Yaskawa INFORM job: KRIS_OTHER_WELDS.JBI

/JOB
//NAME KRIS_OTHER_WELDS
//POS
///NPOS 371,371,371,14,0,0
///TOOL 0
///POSTYPE PULSE
///PULSE
C00000=36471,-76527,-106813,-19264,71481,-77238
C00001=66631,50103,-4762,13566,84527,65375
C00002=104392,-45604,-45068,41730,67848,43971
C00003=102772,-23592,-15673,48581,65359,41958
C00004=103105,-4521,-1193,48225,65783,42370
C00005=103550,-365,5452,48799,64222,41754
C00006=103550,625,8518,49296,63299,41230
C00007=103550,355,7706,49163,63541,41368
C00008=102300,1028,8270,49380,64218,41057
C00009=102134,1217,8640,49454,64220,40967
C00010=102487,1102,8722,49434,63955,41010
C00011=101792,827,6993,49227,64947,41190
C00012=100819,-958,-818,48185,68095,42388
C00013=74228,-100728,-57385,53918,72446,30220
C00014=60504,-146661,-111893,16693,92041,-63510
C00015=81002,-144165,-111893,31958,74905,-63510
C00016=99609,-128801,-101652,29194,69226,-57515
C00017=99609,-127984,-100239,29275,68831,-57620
C00018=99609,-128289,-100766,29244,68978,-57581
C00019=102150,-129321,-101059,28822,67791,-56859
C00020=99944,-132310,-102446,29373,67957,-57721
C00021=94854,-157221,-110079,32013,62771,-61374
C00022=94854,-157221,-110079,32013,62771,-61374
C00023=150575,-180894,-113467,-20602,37776,7473
C00024=131435,-154210,-106652,-7413,43941,-3112
C00025=131414,-154056,-106648,-7392,44016,-3129
C00026=131048,-150684,-105922,-7028,45259,-3400
C00027=131414,-154056,-106648,-7392,44016,-3129
C00028=178670,-106537,-94441,-32173,86364,27351
C00029=174579,-86120,-85943,-32864,94727,28981
C00030=173469,-85635,-85233,-32803,94141,28710
C00031=173469,-85539,-84108,-32766,93596,28870
C00032=173084,-86046,-85408,-32780,93905,28625
C00033=171779,-87936,-86208,-32689,92999,28371
C00034=172551,-86827,-85740,-32743,93534,28522
C00035=185237,-110424,-94728,-32531,92831,33795
C00036=185237,-110424,-94728,-32531,92831,33795
C00037=134012,-175619,-118342,2096,46955,-2797
C00038=133371,-126486,-107062,2327,67886,-2658
C00039=134292,-123400,-104700,2048,67993,-2322
C00040=134292,-122480,-102592,2060,67168,-2335
C00041=134292,-122828,-103379,2055,67474,-2331
C00042=133740,-117277,-101631,2195,69264,-2498
C00043=134292,-122828,-103379,2055,67474,-2331
C00044=145565,-124760,-104669,-1363,67226,1769
C00045=157884,-133264,-102216,-16015,55602,12124
C00046=154931,-135462,-102806,-14939,54301,11078
C00047=159722,-139649,-104449,-17130,54142,13140
C00048=121501,-151260,-116369,16790,67529,-22254
C00049=84851,-125920,-106326,14509,72614,-18670
C00050=87302,-113526,-101119,13757,75261,-17475
C00051=88050,-112106,-100360,13572,75391,-17193
C00052=88050,-111725,-99039,13608,74790,-17261
C00053=88050,-111984,-99928,13584,75193,-17215
C00054=88832,-108808,-98834,13352,75998,-16846
C00055=87807,-112947,-100252,13656,74947,-17329
C00056=92070,-142291,-103311,16392,49176,-14760
C00057=94804,-140634,-102905,14943,49236,-13516
C00058=91121,-138706,-102421,16531,50612,-14939
C00059=93561,-140381,-102567,15560,49394,-14049
C00060=69173,-195704,-118009,34153,38892,-29324
C00061=69173,-195704,-118009,34153,38892,-29324
C00062=107696,-37154,-67359,5229,84713,-5863
C00063=116742,-32674,-55171,12076,80004,-1616
C00064=117154,-30403,-53709,11929,80206,-1458
C00065=117154,-30689,-52627,11956,79411,-1536
C00066=117154,-30552,-53163,11943,79803,-1497
C00067=108517,-16990,-43540,23191,88993,-13455
C00068=109765,-14828,-41918,22897,88763,-13064
C00069=109347,-17906,-44920,22997,89117,-13141
C00070=106896,-6499,-37008,27511,96493,-19470
C00071=107863,-6880,-37313,27352,96184,-19193
C00072=104662,-5505,-36210,27871,97208,-20107
C00073=93389,-55640,-71668,19302,82770,-9184
C00074=93389,-55640,-71668,19302,92834,78584
C00075=111754,-46764,-69921,16160,92456,84768
C00076=113010,-47490,-70150,15902,91999,85126
C00077=113010,-47824,-69220,15892,91281,85034
C00078=113010,-47731,-69491,15895,91487,85061
C00079=112902,-49890,-70751,15912,91185,84985
C00080=100788,-44242,-62951,32464,93570,83345
C00081=95750,-41506,-57227,39958,94516,82624
C00082=97351,-42547,-57870,39748,93692,82997
C00083=107713,-44703,-69881,16984,94226,83661
C00084=110462,-17925,-52010,16025,110800,86473
C00085=112866,-11103,-45097,15475,114636,87689
C00086=116727,-11513,-45414,15662,113935,88992
C00087=102039,-2481,-42089,15122,118996,84328
C00088=102039,-2481,-42089,15122,100704,-14672
C00089=117847,-25402,-50017,12117,83012,-11069
C00090=117859,-24620,-49869,12107,83315,-11036
C00091=117859,-24721,-49537,12111,83065,-11060
C00092=117448,-24507,-49386,12236,83141,-11189
C00093=109902,-9247,-38011,19141,88596,-18895
C00094=104609,19012,-13716,27585,102398,-34238
C00095=104836,21780,-11197,27552,102213,-34199
C00096=98934,25941,-685,39115,101412,-35075
C00097=91600,14785,-13342,39748,106246,-36411
C00098=47111,-89064,-83881,31350,116876,-52529
C00099=81588,-140072,-114826,15376,71241,-20037
C00100=97769,-116268,-100554,7249,70146,-8698
C00101=93709,-113858,-99760,8341,71283,-10082
C00102=110362,-115244,-100357,-6076,70211,7492
C00103=124823,-97243,-93907,-17727,83078,24095
C00104=122674,-104476,-96562,-17426,80631,23684
C00105=131812,-116317,-102091,-19024,80117,27039
C00106=131812,-116317,-102091,-19024,80117,27039
C00107=106372,-151670,-115941,1479,61909,-1124
C00108=97402,-154853,-108420,9880,47553,-8329
C00109=91237,-150897,-107478,16251,51513,-16477
C00110=91228,-148864,-107179,20465,55021,-21052
C00111=78071,-160284,-116606,19433,65818,-26969
C00112=78071,-160284,-116606,19433,65818,-26969
C00113=90794,-133617,-109168,16116,71767,-21274
C00114=92302,-126682,-105486,15702,72721,-20593
C00115=94506,-128481,-105877,15295,71639,-19928
C00116=115362,-143961,-110168,10698,63087,-13119
C00117=118733,-159504,-110501,11315,48800,-13248
C00118=120726,-159269,-110393,10449,48589,-12395
C00119=145117,-154906,-109701,-815,48970,-1768
C00120=160284,-149842,-108565,-14157,53837,11287
C00121=160361,-149780,-108551,-14182,53873,11315
C00122=182605,-105429,-95739,-27625,86741,32308
C00123=182041,-70442,-81142,-28906,106085,40460
C00124=180373,-64217,-77967,-29369,107732,40648
C00125=198406,-78013,-87317,-27723,112552,46613
C00126=172769,-133105,-108161,8035,62165,-26522
C00127=178553,-109735,-99654,-4570,64842,-24680
C00128=178155,-100208,-93897,-4364,66171,-24878
C00129=175286,-95528,-92243,-3183,67417,-25962
C00130=192352,-138021,-108691,-10814,57252,-18824
C00131=195651,-141887,-109704,-12316,56387,-17389
C00132=195651,-141887,-109704,-12316,56387,-17389
C00133=147222,-76033,-86464,7641,74662,-35625
C00134=144580,-61393,-75556,8586,75722,-36452
C00135=156265,-37930,-66612,-3030,87434,-69848
C00136=155034,-33755,-60965,-2668,86065,-70206
C00137=154458,-32798,-60008,-2135,86746,-70342
C00138=155825,-31413,-58479,-2524,86554,-69904
C00139=162790,-57725,-64353,-16754,59169,-66258
C00140=162790,-57725,-64353,-16754,59169,-66258
C00141=155825,-31413,-58479,-2524,86554,-69904
C00142=155825,-31413,-58479,-2524,86554,-69904
C00143=162790,-57725,-64353,-16754,59169,-66258
C00144=165729,-66356,-73131,-18164,60713,-65340
C00145=165729,-63659,-85226,-16965,69151,-66660
C00146=19938,-154159,-115231,-23119,85461,-7967
C00147=13636,-159467,-113845,-12203,49637,-17715
C00148=116484,-130017,-129030,-11526,91164,-19547
C00149=116484,-130017,-129030,-11526,91164,-19547
C00150=101509,-111741,-97351,2474,75173,-11228
C00151=109604,-105261,-90247,737,73969,-8417
C00152=109604,-104665,-88539,738,73224,-8421
C00153=109604,-104936,-89303,737,73555,-8419
C00154=110002,-100393,-87649,645,74866,-8273
C00155=109618,-105123,-90216,732,74019,-8412
C00156=74185,-80593,-80392,7895,82492,-20315
C00157=74487,-79761,-79527,7841,82359,-20221
C00158=74487,-79638,-78308,7850,81677,-20261
C00159=74487,-79693,-78808,7845,81955,-20243
C00160=75396,-77288,-77713,7667,82425,-19905
C00161=74164,-80634,-80212,7899,82363,-20329
C00162=71363,-97810,-96211,8399,83653,-21197
C00163=71363,-97810,-96211,8399,83653,-21197
C00164=75126,-80656,-81685,7709,83157,-19951
C00165=76229,-77543,-78801,7504,82880,-19595
C00166=76229,-77418,-77195,7514,81965,-19651
C00167=76229,-77461,-77677,7510,82237,-19634
C00168=77485,-73926,-76028,7263,82920,-19167
C00169=76229,-77506,-78245,7506,82561,-19615
C00170=111141,-100889,-88631,397,75213,-7875
C00171=111199,-100043,-88075,385,75306,-7854
C00172=111199,-99510,-86287,385,74481,-7854
C00173=111199,-99854,-87425,384,75005,-7852
C00174=111556,-94962,-85553,305,76365,-7724
C00175=110981,-102889,-89081,432,74466,-7929
C00176=63222,-84337,-117253,10216,104159,-22323
C00177=63222,-84337,-117253,10216,104159,-22323
C00178=116461,-126066,-89110,-816,62587,-5937
C00179=121112,-11531,-1732,-22241,71063,6555
C00180=123069,21697,30953,-28709,69461,10931
C00181=122369,24261,34644,-28789,68382,10931
C00182=122349,25171,36872,-28955,67580,11137
C00183=124729,43924,54800,-30715,75908,19671
C00184=123229,45725,56700,-30654,75959,19910
C00185=122369,24261,34644,-28789,68382,10931
C00186=122757,31247,42135,-29026,67616,11292
C00187=122369,32445,43348,-29004,67370,11200
C00188=122776,30953,41451,-28977,67860,11234
C00189=124792,19441,29060,-28915,70056,11467
C00190=123719,29254,39551,-29128,68728,50133
C00191=123432,29487,40138,-29139,68416,50100
C00192=123432,30301,42102,-29286,67723,50287
C00193=123432,29794,40884,-29194,68152,50171
C00194=122305,29700,40790,-29062,67775,49816
C00195=123432,29794,40884,-29194,68152,50171
C00196=130745,-67077,-33050,-30688,66975,53477
C00197=125856,-63248,-28818,-30456,64700,52130
C00198=125856,-62207,-26795,-30622,64084,52309
C00199=125856,-62769,-27883,-30532,64415,52213
C00200=123740,-62907,-27951,-30347,63650,51561
C00201=125856,-63248,-28818,-30456,64700,52130
C00202=154464,-88255,-48627,-31084,74327,60840
C00203=106362,-64202,-67111,7532,73191,-21872
C00204=94843,-131680,-92775,12823,56012,-27739
C00205=140364,-112792,-85989,-36793,59691,-67841
C00206=158545,-73764,-60782,-39609,71363,-63907
C00207=158545,-73538,-60068,-39675,71111,-63809
C00208=158220,-67471,-54290,-39710,70623,-63764
C00209=158220,-67064,-53033,-39832,70183,-63590
C00210=158220,-67225,-53525,-39784,70354,-63658
C00211=159834,-65842,-52837,-39997,71318,-63299
C00212=159834,-65842,-52837,-39997,71318,-63299
C00213=159366,-66137,-52690,-39970,70914,-63355
C00214=160474,-67684,-54367,-40105,71611,-63123
C00215=187581,-124736,-92952,-42921,80369,-54295
C00216=106362,-64202,-67111,7532,73191,-21872
C00217=114111,-33769,-47951,4944,76427,-19032
C00218=116115,-30064,-41477,4332,74239,-18430
C00219=116115,-30038,-40119,4349,73419,-18459
C00220=116091,-30813,-41108,4352,73629,-18459
C00221=116253,-25293,-37304,4290,74115,-18387
C00222=114317,-34919,-41800,5611,66541,-19356
C00223=114260,-33378,-40787,5626,66711,-19367
C00224=115034,-33499,-40868,5308,66647,-19089
C00225=113158,-36981,-44175,6067,67023,-19752
C00226=112664,-46710,-50923,6306,66218,-19974
C00227=89680,-35115,-43687,15042,70735,-27919
C00228=91637,-21855,-35421,13091,75116,-26782
C00229=91876,-20585,-33111,13073,74332,-26785
C00230=91876,-20566,-32258,13104,73831,-26840
C00231=91876,-20585,-33111,13073,74332,-26785
C00232=92389,-17919,-31150,12899,74409,-26598
C00233=92130,-19322,-32180,12987,74366,-26692
C00234=94093,-21573,-33801,12367,73907,-26048
C00235=94752,-22029,-34122,12156,73773,-25827
C00236=94116,-21556,-33780,12360,73899,-26041
C00237=89471,-44398,-62631,13554,80495,-26944
C00238=122819,-38731,-49409,10163,73779,-23755
C00239=123901,-31517,-41329,9859,72397,-23490
C00240=123898,-31367,-41229,9859,72412,-23490
C00241=123846,-28795,-39484,9864,72664,-23488
C00242=122861,-32799,-42184,10217,72396,-23858
C00243=117239,-31881,-41533,12078,73231,-25771
C00244=117050,-26971,-37987,12120,73592,-25801
C00245=117050,-26927,-36697,12165,72838,-25879
C00246=118428,-26989,-37557,11688,73120,-25361
C00247=119059,-27021,-37582,11480,73027,-25151
C00248=118425,-26908,-37435,11691,73088,-25365
C00249=118304,-35951,-45306,11721,73299,-25387
C00250=123411,-39440,-45986,-27831,73569,1045
C00251=123203,-26968,-33658,-27929,72456,1240
C00252=123203,-26817,-32292,-28037,71780,1409
C00253=123203,-26931,-33292,-27958,72274,1285
C00254=123173,-25001,-31943,-27927,72407,1239
C00255=123137,-22619,-30252,-27893,72558,1186
C00256=123207,-27107,-33414,-27962,72262,1288
C00257=122069,-27891,-33955,-27643,71824,948
C00258=121286,-27911,-33965,-27413,71565,701
C00259=122261,-27884,-33947,-27698,71888,1006
C00260=122377,-39377,-48800,-27318,74811,339
C00261=122377,-39377,-48800,-15958,74811,37256
C00262=116853,-24659,-37061,-14175,74133,35375
C00263=116584,-23309,-33957,-14168,72909,35425
C00264=117149,-18043,-30320,-14317,73463,35559
C00265=117861,-38592,-48080,-14522,73947,35755
C00266=104583,-32490,-50397,7546,82362,7604
C00267=105194,-26999,-38249,8695,72546,7274
C00268=107004,-26270,-36315,8108,71553,7839
C00269=105841,-25958,-36017,8513,71647,7439
C00270=93962,-24813,-35260,12474,73301,3377
C00271=93359,-24324,-34888,12668,73417,3175
C00272=84365,-15908,-28760,15403,75492,223
C00273=84333,-15873,-28734,15412,75500,213
C00274=74614,15948,-2221,27741,93727,-20451
C00275=73064,34093,16547,30155,99822,-32312
C00276=73134,34448,17489,31264,97859,-32734
C00277=67749,23419,3523,31459,102357,-33616
C00278=95915,-30118,-44789,16449,81748,-17699
C00279=98720,-22295,-36539,15790,80186,-16929
C00280=100927,-17947,-31539,15262,78961,-16317
C00281=102083,-20206,-33033,12712,77113,-13215
C00282=98715,-18258,-31690,13637,77822,-14313
C00283=114236,-21942,-34401,-8246,75145,9325
C00284=114072,-21865,-34349,-8196,75136,9270
C00285=113262,-31754,-46716,-7868,77565,8837
C00286=121052,-35480,-50751,8872,78740,-8774
C00287=126219,-34781,-43956,7407,74440,-7288
C00288=119242,-20380,-33459,16470,80241,-18104
C00289=118226,-16611,-30649,16706,80643,-18406
C00290=117697,-15053,-29476,16826,80828,-18565
C00291=128590,-25056,-36776,1961,74083,-1425
C00292=133010,-24673,-36504,-4702,74461,5650
C00293=131254,-25215,-36887,-4141,74323,5049
C00294=130676,-43988,-54039,-2112,74946,2871
C00295=144327,-162746,-116257,-7792,53093,8922
C00296=140364,-112792,-85989,-36793,59691,-67841
C00297=158545,-73764,-60782,-39609,71363,-63907
C00298=154861,-52064,-52586,-29243,83996,-69304
C00299=154353,-50613,-51249,-28584,84794,-69672
C00300=152671,-51223,-50857,-28405,83729,-70057
C00301=164464,-77852,-47727,-57510,56856,-52749
C00302=164600,-79193,-48735,-57564,56899,-52688
C00303=152503,-51284,-51279,-28373,83875,-70156
C00304=149379,-69811,-60108,-25771,69929,-67691
C00305=150657,-73399,-57833,-31681,60752,-64672
C00306=164600,-79193,-48735,-57564,56899,-52688
C00307=211845,-135273,-82829,-57573,80898,-40537
C00308=8980,-110764,-82837,-4940,58692,5944
C00309=63222,-84337,-117253,10216,104159,-22323
C00310=63222,-84337,-117253,10216,104159,-22323
C00311=62622,-35658,-60172,17305,99584,-35384
C00312=67983,-29131,-50691,16571,96143,-34035
C00313=68280,-28632,-48929,16503,95291,-34050
C00314=96157,-58786,-67227,12347,86330,-25614
C00315=93243,-56160,-71235,12854,90500,-26173
C00316=74215,-69707,-85545,7852,91184,-19756
C00317=93841,-69746,-85565,-9172,91908,7615
C00318=97380,-51119,-65343,-9768,89472,8971
C00319=98254,-45707,-60597,-9931,89441,9263
C00320=98294,-45060,-62789,-9947,91102,9145
C00321=97224,-52262,-64508,-9752,88371,9004
C00322=70374,-15387,-39875,-4697,89776,63
C00323=72305,-19661,-49372,-5108,93524,541
C00324=103604,-85812,-120886,-11405,106313,9533
C00325=4313,-85812,-120886,-11405,106313,9533
C00326=4313,-85812,-120886,-11405,106313,9533
C00327=116461,-126066,-89110,-816,62587,-5937
C00328=120494,-28298,-18223,-19234,72094,4641
C00329=115081,317,11412,-13994,56205,7379
C00330=111951,8468,21397,-13093,53779,6399
C00331=111881,7001,20107,-13059,53806,6365
C00332=111973,8122,19702,-12964,54626,6300
C00333=115084,14869,27163,-14364,54053,7678
C00334=122843,32694,44412,-26431,63312,23020
C00335=122843,32694,44412,-26431,63312,23020
C00336=126005,74918,92279,-31006,69428,36805
C00337=129411,35206,44111,-29718,78661,35512
C00338=130589,8419,18518,-29555,80810,75073
C00339=123805,36930,48494,-26196,90453,76476
C00340=120628,37037,48526,-26729,89486,75519
C00341=128053,46953,52473,-25525,94200,77226
C00342=132423,-27016,-13437,-24037,82468,48912
C00343=125265,-65617,-33465,-24620,73519,48112
C00344=119787,-70343,-33837,-24664,68336,45094
C00345=120138,-4909,7155,-23652,76131,43583
C00346=120137,-2255,9546,-23662,76032,43605
C00347=120292,48641,58368,-24082,72501,44393
C00348=118376,33653,42209,-20968,68204,36216
C00349=123699,9685,13287,-20232,72289,34129
C00350=136612,-39302,-26410,-22131,74933,38485
C00351=171363,-111780,-58290,-25542,68690,52860
C00352=105993,-174005,-130935,-24309,80821,50388
C00353=106047,-157383,-132399,4283,59082,-17249
C00354=106047,-157383,-132399,4283,59082,-17249
C00355=88146,-87318,-79564,5997,74851,-23158
C00356=100398,-84385,-72843,1794,70423,-11848
C00357=101406,-83692,-71963,1525,70218,-11491
C00358=100271,-90451,-74903,1851,68579,-11922
C00359=100398,-85037,-75228,1783,71555,-11832
C00360=65698,-50267,-54969,10311,79573,-23523
C00361=61954,-58139,-63827,11098,81445,-24649
C00362=56555,-47628,-57747,17133,88641,-29036
C00363=60241,-40499,-49477,16589,86520,-28045
C00364=90516,-77386,-69324,11133,74773,-18779
C00365=88053,-87457,-77735,11673,75122,-19621
C00366=72402,-151240,-127472,14898,75587,-25161
C00367=72402,-151240,-127472,14898,75587,-25161
C00368=-10,-151240,-127472,4482,80219,-3882
C00369=36471,-76527,-106813,-19264,71481,-77238
C00370=36471,-76527,-106813,-19264,71481,-77238
BC00000=295309,515546,1075134
BC00001=156427,631939,1073423
BC00002=296646,526466,1071703
BC00003=296646,526466,1071703
BC00004=296646,526466,1071703
BC00005=296646,526466,1071703
BC00006=296646,526466,1071703
BC00007=296646,526466,1071703
BC00008=296646,526466,1071703
BC00009=296646,526466,1071703
BC00010=296645,526465,1071702
BC00011=296645,526465,1071702
BC00012=296645,526465,1071702
BC00013=296645,526465,1071702
BC00014=41422,444909,146072
BC00015=41422,407031,82823
BC00016=41422,407031,82823
BC00017=41422,407031,82823
BC00018=41422,407031,82823
BC00019=41422,407031,82823
BC00020=41422,407031,82823
BC00021=41422,407031,82823
BC00022=102400,418935,82823
BC00023=102400,418935,82823
BC00024=102400,418935,82823
BC00025=102400,418935,82823
BC00026=102400,418935,82823
BC00027=102400,418935,82823
BC00028=102400,418935,82823
BC00029=102400,418935,82821
BC00030=102400,418935,82821
BC00031=102400,418935,82821
BC00032=102400,418935,82821
BC00033=102400,418935,82821
BC00034=102400,418935,82821
BC00035=102400,418935,82821
BC00036=359098,418935,82821
BC00037=359098,418935,82821
BC00038=359098,418935,82821
BC00039=359098,418935,82821
BC00040=359098,418935,82821
BC00041=359098,418935,82821
BC00042=359098,418935,82821
BC00043=359098,418935,82821
BC00044=359098,418935,82821
BC00045=359098,418935,82821
BC00046=359098,418935,82821
BC00047=359098,418935,82821
BC00048=359098,418935,82821
BC00049=359098,418935,82821
BC00050=359098,418935,82821
BC00051=359098,418935,82821
BC00052=359098,418935,82821
BC00053=359098,418935,82821
BC00054=359098,418935,82821
BC00055=359098,418935,82821
BC00056=359098,418935,82821
BC00057=359098,418935,82821
BC00058=359098,418935,82821
BC00059=359098,418935,82821
BC00060=359098,418935,82821
BC00061=396081,492115,577151
BC00062=396081,492115,759834
BC00063=396081,492115,759834
BC00064=396081,492115,759834
BC00065=396081,492115,759834
BC00066=396081,492115,759834
BC00067=396081,492115,759834
BC00068=396081,492115,759834
BC00069=396081,492115,759834
BC00070=396081,492115,759834
BC00071=396081,492115,759834
BC00072=396081,492115,759834
BC00073=396081,492115,759834
BC00074=396081,492115,759834
BC00075=396081,492115,759834
BC00076=396081,492115,759834
BC00077=396081,492115,759834
BC00078=396081,492115,759834
BC00079=396081,492115,759834
BC00080=396081,492115,759834
BC00081=396081,492115,759834
BC00082=396081,492115,759834
BC00083=396081,492115,759834
BC00084=396081,492114,759833
BC00085=396081,492114,759833
BC00086=396081,492114,759833
BC00087=396081,492114,759833
BC00088=396081,492114,759833
BC00089=396081,492114,759833
BC00090=396081,492114,759833
BC00091=396081,492114,759833
BC00092=396081,492114,759833
BC00093=396081,492114,759833
BC00094=396081,492114,759833
BC00095=396081,492114,759833
BC00096=396081,492114,759833
BC00097=396081,492114,759833
BC00098=396081,492114,759833
BC00099=359098,418935,82821
BC00100=359098,418935,82821
BC00101=359098,418935,82821
BC00102=359098,418935,82821
BC00103=359098,418935,82821
BC00104=359098,418935,82821
BC00105=359098,418935,82821
BC00106=308682,418935,82821
BC00107=314094,408245,75283
BC00108=314839,406777,74246
BC00109=314838,406775,74246
BC00110=314838,406775,74246
BC00111=314838,406775,74246
BC00112=121869,406775,74246
BC00113=121869,406775,74246
BC00114=121869,406775,74246
BC00115=121869,406775,74246
BC00116=121869,406775,74246
BC00117=121869,406775,74246
BC00118=121869,406775,74246
BC00119=121869,406775,74246
BC00120=121869,406775,74246
BC00121=121869,406775,74246
BC00122=121869,406775,74246
BC00123=121869,406775,74246
BC00124=121869,406775,74246
BC00125=121869,406775,74246
BC00126=121869,406775,74246
BC00127=121869,406775,74246
BC00128=121869,406775,74246
BC00129=121869,406775,74246
BC00130=121869,406775,74246
BC00131=269123,509849,222924
BC00132=368825,466980,895939
BC00133=368824,466980,895938
BC00134=368824,466980,895938
BC00135=368824,466980,895938
BC00136=368824,466980,895938
BC00137=368824,466980,895938
BC00138=368824,466980,895938
BC00139=368824,466980,895938
BC00140=368824,466980,900103
BC00141=368824,466980,902063
BC00142=368824,466980,895938
BC00143=368824,466980,895938
BC00144=368824,466980,895938
BC00145=368824,466980,895938
BC00146=323528,523697,663885
BC00147=215457,510863,1034966
BC00148=215457,510863,1061671
BC00149=302533,388804,1061671
BC00150=302533,388804,1022471
BC00151=302533,388804,1022471
BC00152=302533,388804,1022471
BC00153=302533,388804,1022471
BC00154=302533,388804,1022471
BC00155=302533,388804,1022471
BC00156=302533,388804,1022471
BC00157=302533,388804,1022471
BC00158=302533,388804,1022471
BC00159=302533,388804,1022471
BC00160=302533,388804,1022471
BC00161=302533,388804,1022471
BC00162=291893,393028,1023549
BC00163=48415,393028,1023549
BC00164=48415,393028,1023549
BC00165=48415,393028,1023549
BC00166=48415,393028,1023549
BC00167=48415,393028,1023549
BC00168=48415,393028,1023549
BC00169=48415,393028,1023549
BC00170=48415,393028,1023549
BC00171=48415,393028,1023549
BC00172=48415,393028,1023549
BC00173=48415,393028,1023549
BC00174=48415,393028,1023549
BC00175=48415,393028,1023549
BC00176=48415,393028,1023549
BC00177=21675,516959,1023549
BC00178=1991,516959,1023549
BC00179=1992,516959,1023547
BC00180=1992,516959,1023546
BC00181=1992,516959,1023546
BC00182=1992,516959,1023546
BC00183=1992,516959,1023546
BC00184=1992,516959,1023546
BC00185=1992,516959,1023546
BC00186=1992,516959,1023546
BC00187=1992,516959,1023546
BC00188=1992,516959,1023546
BC00189=1992,516959,1023546
BC00190=1992,516959,1023543
BC00191=1992,516959,1023543
BC00192=1992,516959,1023543
BC00193=1992,516959,1023543
BC00194=1992,516959,1023543
BC00195=1992,516959,1023543
BC00196=1992,516959,1023543
BC00197=1992,516959,1023543
BC00198=1992,516959,1023543
BC00199=1992,516959,1023543
BC00200=1992,516959,1023543
BC00201=1992,516959,1023543
BC00202=1992,516959,1023543
BC00203=48415,502452,196482
BC00204=170464,492672,1002532
BC00205=170463,451272,1002531
BC00206=170463,451272,1002531
BC00207=170463,451272,1002531
BC00208=170463,451272,1002531
BC00209=170463,451272,1002531
BC00210=170463,451272,1002531
BC00211=170463,451272,1002531
BC00212=170463,451272,1002531
BC00213=170463,451272,1002531
BC00214=170463,451272,1002531
BC00215=170463,451272,1002531
BC00216=48415,502452,196482
BC00217=48415,502452,196482
BC00218=48415,502452,196482
BC00219=48415,502452,196482
BC00220=48415,502452,196482
BC00221=48415,502452,196482
BC00222=48415,502452,196482
BC00223=48415,502452,196482
BC00224=48415,502452,196482
BC00225=48415,502452,196482
BC00226=48415,502452,196482
BC00227=48415,502452,196482
BC00228=48415,502452,196482
BC00229=48415,502452,196480
BC00230=48415,502452,196480
BC00231=48415,502452,196480
BC00232=48415,502452,196480
BC00233=48415,502452,196480
BC00234=48415,502452,196480
BC00235=48415,502452,196480
BC00236=48415,502452,196480
BC00237=48415,502452,196480
BC00238=376815,502452,196479
BC00239=376815,502452,196479
BC00240=376815,502452,196479
BC00241=376815,502452,196479
BC00242=376815,502452,196479
BC00243=376815,502452,196479
BC00244=376815,502452,196479
BC00245=376815,502452,196479
BC00246=376815,502452,196479
BC00247=376815,502452,196479
BC00248=376815,502452,196479
BC00249=376815,502452,196479
BC00250=376815,502452,196479
BC00251=376815,502452,196479
BC00252=376815,502452,196479
BC00253=376815,502452,196479
BC00254=376815,502452,196479
BC00255=376815,502452,196479
BC00256=376815,502452,196479
BC00257=376815,502452,196479
BC00258=376815,502452,196479
BC00259=376815,502452,196479
BC00260=376815,502452,196479
BC00261=376815,502452,196479
BC00262=376815,502452,196477
BC00263=376815,502452,196477
BC00264=376815,502452,196477
BC00265=376815,502452,196477
BC00266=271956,502452,196471
BC00267=271956,502452,196471
BC00268=271956,502452,196471
BC00269=271956,502452,196471
BC00270=271956,502452,196471
BC00271=271956,502452,196471
BC00272=271956,502452,196471
BC00273=271956,502452,196471
BC00274=271956,502452,196471
BC00275=271956,502452,196471
BC00276=271956,502452,196471
BC00277=271956,502452,196471
BC00278=72152,502452,196464
BC00279=72152,502452,196464
BC00280=72152,502452,196462
BC00281=72152,502452,196462
BC00282=72152,502452,196462
BC00283=72152,502452,196460
BC00284=72152,502452,196460
BC00285=72152,502452,196460
BC00286=72152,502452,196463
BC00287=72153,502452,196461
BC00288=72153,502452,196461
BC00289=72153,502452,196461
BC00290=72153,502452,196461
BC00291=72153,502452,196461
BC00292=72153,502452,196461
BC00293=72153,502452,196461
BC00294=72153,502452,196461
BC00295=130981,502452,956451
BC00296=170463,451272,1002531
BC00297=170463,451272,1002531
BC00298=170463,451272,1002531
BC00299=170463,451272,1002531
BC00300=170463,451272,1002531
BC00301=170463,451272,1002531
BC00302=170463,451272,1002531
BC00303=170463,451272,1002531
BC00304=170463,451272,1002531
BC00305=170463,451272,1002531
BC00306=170463,451272,1002531
BC00307=170463,451272,1002531
BC00308=72153,524540,501815
BC00309=21675,516959,1023549
BC00310=31843,416781,1023549
BC00311=31843,416781,1023544
BC00312=31843,416781,1023544
BC00313=31843,416781,1023541
BC00314=31842,416781,1023535
BC00315=31842,416781,1023535
BC00316=31843,416781,1023549
BC00317=239078,416781,1023549
BC00318=239078,416781,1023549
BC00319=239078,416781,1023547
BC00320=239078,416781,1023547
BC00321=239078,416781,1023547
BC00322=239078,416781,1023547
BC00323=239078,416781,1023547
BC00324=239078,416781,1023547
BC00325=178913,503823,1023547
BC00326=46741,503823,1023547
BC00327=1991,516959,1023549
BC00328=1992,516958,1023545
BC00329=1993,516957,1023537
BC00330=1993,516957,1023537
BC00331=1993,516957,1023537
BC00332=1993,516957,1023537
BC00333=1993,516957,1023537
BC00334=1993,516957,1023537
BC00335=1993,516957,1023537
BC00336=1993,516957,1023537
BC00337=1993,516957,1023537
BC00338=1993,516957,1023537
BC00339=1993,516957,1023537
BC00340=1993,516957,1023537
BC00341=1993,516957,1023537
BC00342=1993,516957,1023537
BC00343=1993,516957,1023537
BC00344=1993,516957,1023537
BC00345=1993,516957,1023537
BC00346=1993,516957,1023537
BC00347=1993,516957,1023537
BC00348=1993,516957,1023537
BC00349=1993,516957,1023537
BC00350=1993,516957,1023537
BC00351=1993,510926,1023537
BC00352=1993,470129,1066426
BC00353=1993,470129,1066426
BC00354=84610,404458,1066426
BC00355=84610,404458,1066426
BC00356=84610,404458,1066426
BC00357=84610,404458,1066426
BC00358=84610,404458,1066426
BC00359=84610,404458,1066426
BC00360=84610,404458,1066426
BC00361=84610,404458,1066426
BC00362=211915,404458,1066426
BC00363=211915,404458,1066426
BC00364=211915,404458,1066426
BC00365=211915,404458,1066426
BC00366=211915,397838,1066426
BC00367=211915,487640,1066426
BC00368=211915,519572,1065201
BC00369=295309,515546,1075134
BC00370=295309,515546,1075134
EC00000=1596315,-183832
EC00001=1596314,-183833
EC00002=1596315,-183832
EC00003=1596315,-183832
EC00004=1596315,-183832
EC00005=1596315,-183832
EC00006=1596315,-183832
EC00007=1596315,-183832
EC00008=1596315,-183832
EC00009=1596315,-183832
EC00010=1596315,-183832
EC00011=1596315,-183832
EC00012=1596315,-183832
EC00013=1596315,-183832
EC00014=1596315,-183832
EC00015=1596315,-183832
EC00016=1596315,-183832
EC00017=1596315,-183832
EC00018=1596315,-183832
EC00019=1596315,-183832
EC00020=1596315,-183832
EC00021=1596315,-183832
EC00022=1596315,-183832
EC00023=1596315,-183832
EC00024=1596315,-183832
EC00025=1596315,-183832
EC00026=1596315,-183832
EC00027=1596315,-183832
EC00028=1596315,-183832
EC00029=1596315,-183832
EC00030=1596315,-183832
EC00031=1596315,-183832
EC00032=1596315,-183832
EC00033=1596315,-183832
EC00034=1596315,-183832
EC00035=1596315,-183832
EC00036=1596315,-183832
EC00037=1596315,-183832
EC00038=1596315,-183832
EC00039=1596315,-183832
EC00040=1596315,-183832
EC00041=1596315,-183832
EC00042=1596315,-183832
EC00043=1596315,-183832
EC00044=1596315,-183832
EC00045=1596315,-183832
EC00046=1596315,-183832
EC00047=1596315,-183832
EC00048=1596315,-183832
EC00049=1596315,-183832
EC00050=1596315,-183832
EC00051=1596315,-183832
EC00052=1596315,-183832
EC00053=1596315,-183832
EC00054=1596315,-183832
EC00055=1596315,-183832
EC00056=1596315,-183832
EC00057=1596315,-183832
EC00058=1596315,-183832
EC00059=1596315,-183832
EC00060=1596315,-183832
EC00061=1596315,-183832
EC00062=1863244,361735
EC00063=1863244,361735
EC00064=1863244,361735
EC00065=1863244,361735
EC00066=1863244,361735
EC00067=1863244,361735
EC00068=1863244,361735
EC00069=1863244,361735
EC00070=1863244,361735
EC00071=1863244,361735
EC00072=1863244,361735
EC00073=1863244,361735
EC00074=1863244,361735
EC00075=1863244,361735
EC00076=1863244,361735
EC00077=1863244,361735
EC00078=1863244,361735
EC00079=1863244,361735
EC00080=1863244,361735
EC00081=1863244,361735
EC00082=1863244,361735
EC00083=1863244,361735
EC00084=1863245,361734
EC00085=1863246,361734
EC00086=1863246,361734
EC00087=1863246,361734
EC00088=1863246,361734
EC00089=1863246,361734
EC00090=1863246,361734
EC00091=1863246,361734
EC00092=1863246,361734
EC00093=1863246,361734
EC00094=1863246,361734
EC00095=1863246,361734
EC00096=1863246,361734
EC00097=1863246,361734
EC00098=1863246,361734
EC00099=1596315,-183832
EC00100=1596315,-183832
EC00101=1596315,-183832
EC00102=1596315,-183832
EC00103=1596315,-183832
EC00104=1596315,-183832
EC00105=1596315,-183832
EC00106=1596315,-183832
EC00107=1596315,-183832
EC00108=1596315,-183832
EC00109=1596315,-183832
EC00110=1596315,-183832
EC00111=1596315,-183832
EC00112=1596315,-183832
EC00113=1596315,-183832
EC00114=1596315,-183832
EC00115=1596315,-183832
EC00116=1596315,-183832
EC00117=1596315,-183832
EC00118=1596315,-183832
EC00119=1596315,-183832
EC00120=1596315,-183832
EC00121=1596315,-183832
EC00122=1596315,-183832
EC00123=1596315,-183832
EC00124=1596315,-183832
EC00125=1596315,-183832
EC00126=1596315,-183832
EC00127=1596315,-183832
EC00128=1596315,-183832
EC00129=1596315,-183832
EC00130=1596315,-183832
EC00131=1596315,-183832
EC00132=1596315,-183832
EC00133=1596317,-183832
EC00134=1596317,-183832
EC00135=1596317,-183832
EC00136=1596317,-183832
EC00137=1596317,-183832
EC00138=1596317,-183832
EC00139=1596317,-183832
EC00140=1596317,-183832
EC00141=1596317,-183832
EC00142=1596317,-183832
EC00143=1596317,-183832
EC00144=1596317,-183832
EC00145=1596317,-183832
EC00146=1596882,372644
EC00147=1857823,372644
EC00148=1857823,372644
EC00149=1857823,372644
EC00150=1857823,372644
EC00151=1857823,372644
EC00152=1857823,372644
EC00153=1857823,372644
EC00154=1857823,372644
EC00155=1857823,372644
EC00156=1857823,372644
EC00157=1857823,372644
EC00158=1857823,372644
EC00159=1857823,372644
EC00160=1857823,372644
EC00161=1857823,372644
EC00162=1857823,372644
EC00163=1857823,372644
EC00164=1857823,372644
EC00165=1857823,372644
EC00166=1857823,372644
EC00167=1857823,372644
EC00168=1857823,372644
EC00169=1857823,372644
EC00170=1857823,372644
EC00171=1857823,372644
EC00172=1857823,372644
EC00173=1857823,372644
EC00174=1857823,372644
EC00175=1857823,372644
EC00176=1857823,372644
EC00177=1857823,372644
EC00178=1857823,372644
EC00179=1857824,372644
EC00180=1857824,372644
EC00181=1857824,372644
EC00182=1857824,372644
EC00183=1857824,372644
EC00184=1857824,372644
EC00185=1857824,372644
EC00186=1857824,372644
EC00187=1857824,372644
EC00188=1857824,372644
EC00189=1857824,372644
EC00190=1857824,372644
EC00191=1857824,372644
EC00192=1857824,372644
EC00193=1857824,372644
EC00194=1857824,372644
EC00195=1857824,372644
EC00196=1857824,372644
EC00197=1857824,372644
EC00198=1857824,372644
EC00199=1857824,372644
EC00200=1857824,372644
EC00201=1857824,372644
EC00202=1857824,372644
EC00203=1596314,929120
EC00204=1596314,929120
EC00205=1596314,929119
EC00206=1596314,929119
EC00207=1596314,929119
EC00208=1596314,929119
EC00209=1596314,929119
EC00210=1596314,929119
EC00211=1596314,929119
EC00212=1596314,929119
EC00213=1596314,929119
EC00214=1596314,929119
EC00215=1596314,929119
EC00216=1596314,929120
EC00217=1596314,929120
EC00218=1596314,929120
EC00219=1596314,929120
EC00220=1596314,929120
EC00221=1596314,929120
EC00222=1596314,929120
EC00223=1596314,929120
EC00224=1596314,929120
EC00225=1596314,929120
EC00226=1596314,929120
EC00227=1596314,929120
EC00228=1596314,929120
EC00229=1596314,929119
EC00230=1596314,929119
EC00231=1596314,929119
EC00232=1596314,929119
EC00233=1596314,929119
EC00234=1596314,929119
EC00235=1596314,929119
EC00236=1596314,929119
EC00237=1596314,929119
EC00238=1596314,929119
EC00239=1596314,929119
EC00240=1596314,929119
EC00241=1596314,929119
EC00242=1596314,929119
EC00243=1596314,929119
EC00244=1596314,929119
EC00245=1596314,929119
EC00246=1596314,929119
EC00247=1596314,929119
EC00248=1596314,929119
EC00249=1596314,929119
EC00250=1596314,929119
EC00251=1596314,929119
EC00252=1596314,929119
EC00253=1596314,929119
EC00254=1596314,929119
EC00255=1596314,929119
EC00256=1596314,929119
EC00257=1596314,929119
EC00258=1596314,929119
EC00259=1596314,929119
EC00260=1596314,929119
EC00261=1596314,929119
EC00262=1596314,929119
EC00263=1596314,929119
EC00264=1596314,929119
EC00265=1596314,929119
EC00266=1596314,929119
EC00267=1596314,929119
EC00268=1596314,929119
EC00269=1596314,929119
EC00270=1596314,929119
EC00271=1596314,929119
EC00272=1596314,929119
EC00273=1596314,929119
EC00274=1596314,929119
EC00275=1596314,929119
EC00276=1596314,929119
EC00277=1596314,929119
EC00278=1596314,929119
EC00279=1596314,929119
EC00280=1596314,929119
EC00281=1596314,929119
EC00282=1596314,929119
EC00283=1596314,929119
EC00284=1596314,929119
EC00285=1596314,929119
EC00286=1596314,929119
EC00287=1596314,929119
EC00288=1596314,929119
EC00289=1596314,929119
EC00290=1596314,929119
EC00291=1596314,929119
EC00292=1596314,929119
EC00293=1596314,929119
EC00294=1596314,929119
EC00295=1596314,929119
EC00296=1596314,929119
EC00297=1596314,929119
EC00298=1596314,929118
EC00299=1596314,929118
EC00300=1596314,929118
EC00301=1596314,929118
EC00302=1596314,929118
EC00303=1596314,929118
EC00304=1596314,929118
EC00305=1596314,929118
EC00306=1596314,929118
EC00307=1596314,929118
EC00308=1596314,929119
EC00309=1857823,372644
EC00310=1857823,372644
EC00311=1857825,372644
EC00312=1857825,372644
EC00313=1857826,372644
EC00314=1857827,372644
EC00315=1857827,372644
EC00316=1857823,372644
EC00317=1857823,372644
EC00318=1857823,372644
EC00319=1857824,372644
EC00320=1857824,372644
EC00321=1857824,372644
EC00322=1857824,372644
EC00323=1857824,372644
EC00324=1857824,372644
EC00325=1857824,372644
EC00326=1857824,372644
EC00327=1857823,372644
EC00328=1857824,372644
EC00329=1857827,372644
EC00330=1857827,372644
EC00331=1857827,372644
EC00332=1857827,372644
EC00333=1857827,372644
EC00334=1857827,372644
EC00335=1857827,372644
EC00336=1857827,372644
EC00337=1857827,372644
EC00338=1857827,372644
EC00339=1857827,372644
EC00340=1857827,372644
EC00341=1857827,372644
EC00342=1857827,372644
EC00343=1857827,372644
EC00344=1857827,372644
EC00345=1857827,372644
EC00346=1857827,372644
EC00347=1857827,372644
EC00348=1857827,372644
EC00349=1857827,372644
EC00350=1857827,372644
EC00351=1857827,372644
EC00352=1857827,372644
EC00353=1857827,372644
EC00354=1857827,372644
EC00355=1857827,372644
EC00356=1857827,372644
EC00357=1857827,372644
EC00358=1857827,372644
EC00359=1857827,372644
EC00360=1857827,372644
EC00361=1857827,372644
EC00362=1857827,372644
EC00363=1857827,372644
EC00364=1857827,372644
EC00365=1857827,372644
EC00366=1857827,372644
EC00367=1857827,372644
EC00368=1857827,372644
EC00369=1596315,-183832
EC00370=0,-183832
///POSTYPE BASE
///RECTAN
///RCONF 0,0,0,0,1,0,0,0,0,0,0,0,0,0,0,0,0,0,0,0,0,0,0,0
P00006=2.006,1.622,-0.565,0.0000,0.0000,0.0000
P00021=0.073,2.058,-0.109,0.0000,0.0000,0.0000
P00022=2.006,1.622,-0.565,0.0000,0.0000,0.0000
///RCONF 0,0,0,0,0,0,0,0,0,0,0,0,0,0,0,0,0,0,0,0,0,0,0,0
P00023=-2.957,-4.083,2.762,0.0000,0.0000,0.0000
P00024=-1.466,-0.226,-0.419,0.0000,0.0000,0.0000
P00025=3.643,0.007,-2.585,0.0000,0.0000,0.0000
P00026=2.644,0.055,-2.583,0.0000,0.0000,0.0000
P00027=2.278,0.099,-4.210,0.0000,0.0000,0.0000
P00028=-1.778,-0.182,-2.050,0.0000,0.0000,0.0000
P00030=-0.014,-0.768,0.131,0.0000,0.0000,0.0000
P00031=-0.170,0.039,-0.647,0.0000,0.0000,0.0000
P00032=-0.423,0.157,3.222,0.0000,0.0000,0.0000
P00071=-2.048,-0.034,-9.092,0.0000,0.0000,0.0000
P00072=-1.595,-0.049,-6.373,0.0000,0.0000,0.0000
//INST
///DATE 2024/12/19 20:01
///ATTR SC,RW
///GROUP1 RB1,BS1
///GROUP2 ST1
NOP
MOVJ C00000 BC00000 VJ=100.00  +MOVJ EC00000 VJ=100.00
CALL JOB:CLEAN-R1_KM_NEW
MOVJ C00001 BC00001 VJ=100.00  +MOVJ EC00001 VJ=100.00
MOVJ C00002 BC00002 VJ=100.00  +MOVJ EC00002 VJ=100.00
MOVJ C00003 BC00003 VJ=100.00  +MOVJ EC00003 VJ=100.00
SMOVL C00004 BC00004 V=400.0  +MOVJ EC00004
SFTOF3D
SMOVL C00005 BC00005 V=100.0  +MOVJ EC00005
SREFP 3 C00006 BC00006  +REFP EC00006
CALL JOB:SEARCH-R1-S13D
SET P071 P006
SFTON3D P071
SMOVL C00007 BC00007 V=100.0  +MOVJ EC00007
SMOVL C00008 BC00008 V=100.0  +MOVJ EC00008
SMOVL C00009 BC00009 V=83.3 PL=0  +MOVJ EC00009
SREFP 3 C00010 BC00010  +REFP EC00010
CALL JOB:SEARCH-R1-S13D
SET P071 P006
SFTON3D P071
SMOVL C00011 BC00011 V=100.0  +MOVJ EC00011
SFTOF3D
SMOVL C00012 BC00012 V=1000.0  +MOVJ EC00012
SMOVL C00013 BC00013 V=1000.0  +MOVJ EC00013
MOVJ C00014 BC00014 VJ=100.00  +MOVJ EC00014 VJ=100.00
MOVJ C00015 BC00015 VJ=100.00  +MOVJ EC00015 VJ=100.00
'SE1
SMOVL C00016 BC00016 V=100.0  +MOVJ EC00016
SREFP 3 C00017 BC00017  +REFP EC00017
CALL JOB:SEARCH-R1-S13D
SET P021 P006
SFTON3D P021
SMOVL C00018 BC00018 V=100.0  +MOVJ EC00018
SREFP 3 C00019 BC00019  +REFP EC00019
CALL JOB:SEARCH-R1-S13D
SET P021 P006
SFTON3D P021
SMOVL C00020 BC00020 V=100.0  +MOVJ EC00020
SFTOF3D
MOVJ C00021 BC00021 VJ=100.00  +MOVJ EC00021 VJ=100.00
MOVJ C00022 BC00022 VJ=100.00  +MOVJ EC00022 VJ=100.00
MOVJ C00023 BC00023 VJ=100.00  +MOVJ EC00023 VJ=100.00
MOVJ C00024 BC00024 VJ=100.00  +MOVJ EC00024 VJ=100.00
SFTOF3D
SMOVL C00025 BC00025 V=100.0  +MOVJ EC00025
SREFP 3 C00026 BC00026  +REFP EC00026
CALL JOB:SEARCH-R1-S13D
SET P022 P006
SFTON3D P022
SMOVL C00027 BC00027 V=100.0  +MOVJ EC00027
MOVJ C00028 BC00028 VJ=60.00  +MOVJ EC00028 VJ=100.00
MOVJ C00029 BC00029 VJ=60.00  +MOVJ EC00029 VJ=100.00
SMOVL C00030 BC00030 V=100.0  +MOVJ EC00030
SREFP 3 C00031 BC00031  +REFP EC00031
CALL JOB:SEARCH-R1-S13D
SET P022 P006
SFTON3D P022
SMOVL C00032 BC00032 V=100.0  +MOVJ EC00032
SREFP 3 C00033 BC00033  +REFP EC00033
CALL JOB:SEARCH-R1-S13D
SET P022 P006
SFTON3D P022
SMOVL C00034 BC00034 V=100.0  +MOVJ EC00034
SFTOF3D
'SE2
MOVJ C00035 BC00035 VJ=100.00  +MOVJ EC00035 VJ=100.00
MOVJ C00036 BC00036 VJ=100.00  +MOVJ EC00036 VJ=100.00
MOVJ C00037 BC00037 VJ=100.00  +MOVJ EC00037 VJ=100.00
MOVJ C00038 BC00038 VJ=100.00  +MOVJ EC00038 VJ=100.00
SMOVL C00039 BC00039 V=100.0  +MOVJ EC00039
SREFP 3 C00040 BC00040  +REFP EC00040
CALL JOB:SEARCH-R1-S13D
SET P023 P006
SFTON3D P023
SMOVL C00041 BC00041 V=100.0  +MOVJ EC00041
SREFP 3 C00042 BC00042  +REFP EC00042
CALL JOB:SEARCH-R1-S13D
SET P023 P006
SFTON3D P023
SMOVL C00043 BC00043 V=100.0  +MOVJ EC00043
SMOVL C00044 BC00044 V=100.0  +MOVJ EC00044
SMOVL C00045 BC00045 V=100.0  +MOVJ EC00045
SREFP 3 C00046 BC00046  +REFP EC00046
CALL JOB:SEARCH-R1-S13D
SET P023 P006
SFTON3D P023
SMOVL C00047 BC00047 V=100.0  +MOVJ EC00047
SFTOF3D
'SE3
MOVJ C00048 BC00048 VJ=100.00  +MOVJ EC00048 VJ=100.00
MOVJ C00049 BC00049 VJ=100.00  +MOVJ EC00049 VJ=100.00
MOVJ C00050 BC00050 VJ=100.00  +MOVJ EC00050 VJ=100.00
'SE4
SMOVL C00051 BC00051 V=100.0  +MOVJ EC00051
SREFP 3 C00052 BC00052  +REFP EC00052
CALL JOB:SEARCH-R1-S13D
SET P024 P006
SFTON3D P024
SMOVL C00053 BC00053 V=100.0  +MOVJ EC00053
SREFP 3 C00054 BC00054  +REFP EC00054
CALL JOB:SEARCH-R1-S13D
SET P024 P006
SFTON3D P024
SMOVL C00055 BC00055 V=100.0  +MOVJ EC00055
MOVJ C00056 BC00056 VJ=100.00  +MOVJ EC00056 VJ=100.00
SMOVL C00057 BC00057 V=100.0  +MOVJ EC00057
SREFP 3 C00058 BC00058  +REFP EC00058
CALL JOB:SEARCH-R1-S13D
SET P024 P006
SFTON3D P024
SMOVL C00059 BC00059 V=100.0  +MOVJ EC00059
SFTOF3D
MOVJ C00060 BC00060 VJ=100.00  +MOVJ EC00060 VJ=100.00
MOVJ C00061 BC00061 VJ=100.00  +MOVJ EC00061 VJ=100.00
MOVJ C00062 BC00062 VJ=100.00  +MOVJ EC00062 VJ=100.00
MOVJ C00063 BC00063 VJ=100.00  +MOVJ EC00063 VJ=100.00
'SE5
SMOVL C00064 BC00064 V=100.0  +MOVJ EC00064
SREFP 3 C00065 BC00065  +REFP EC00065
CALL JOB:SEARCH-R1-S13D
SET P025 P006
SFTON3D P025
SMOVL C00066 BC00066 V=100.0  +MOVJ EC00066
SMOVL C00067 BC00067 V=100.0  +MOVJ EC00067
SREFP 3 C00068 BC00068  +REFP EC00068
CALL JOB:SEARCH-R1-S13D
SET P025 P006
SFTON3D P025
SMOVL C00069 BC00069 V=100.0  +MOVJ EC00069
SMOVL C00070 BC00070 V=100.0  +MOVJ EC00070
SREFP 3 C00071 BC00071  +REFP EC00071
CALL JOB:SEARCH-R1-S13D
SET P025 P006
SFTON3D P025
SMOVL C00072 BC00072 V=100.0  +MOVJ EC00072
SFTOF3D
MOVJ C00073 BC00073 VJ=100.00  +MOVJ EC00073 VJ=100.00
MOVJ C00074 BC00074 VJ=100.00  +MOVJ EC00074 VJ=100.00
MOVJ C00075 BC00075 VJ=100.00  +MOVJ EC00075 VJ=100.00
'SE6
SMOVL C00076 BC00076 V=100.0  +MOVJ EC00076
SREFP 3 C00077 BC00077  +REFP EC00077
CALL JOB:SEARCH-R1-S13D
SET P026 P006
SFTON3D P026
SMOVL C00078 BC00078 V=100.0  +MOVJ EC00078
SREFP 3 C00079 BC00079  +REFP EC00079
CALL JOB:SEARCH-R1-S13D
SET P026 P006
SFTON3D P026
SMOVL C00080 BC00080 V=100.0  +MOVJ EC00080
SMOVL C00081 BC00081 V=100.0  +MOVJ EC00081
SREFP 3 C00082 BC00082  +REFP EC00082
CALL JOB:SEARCH-R1-S13D
SET P026 P006
SFTON3D P026
SMOVL C00083 BC00083 V=100.0  +MOVJ EC00083
MOVJ C00084 BC00084 VJ=15.00  +MOVJ EC00084 VJ=10.00
MACRO1 MJ#(0) ARGF14
SMOVL C00085 BC00085 V=250.0 PL=0  +MOVJ EC00085
ARCON
SWVON WEV#(66)
SMOVL C00086 BC00086 V=8.3  +MOVJ EC00086
ARCOF
SWVOF
SFTOF3D
MOVJ C00087 BC00087 VJ=30.00  +MOVJ EC00087 VJ=15.00
MOVJ C00088 BC00088 VJ=100.00  +MOVJ EC00088 VJ=100.00
MACRO1 MJ#(0) ARGF9
SFTON3D P025
SREFP 1 C00089 BC00089  +REFP EC00089
SREFP 2 C00090 BC00090  +REFP EC00090
SMOVL C00091 BC00091 V=250.0 PL=0  +MOVJ EC00091
ARCON
SWVON WEV#(68)
SMOVL C00092 BC00092 V=7.5  +MOVJ EC00092
SMOVL C00093 BC00093 V=7.5  +MOVJ EC00093
SMOVL C00094 BC00094 V=10.8  +MOVJ EC00094
SMOVL C00095 BC00095 V=10.8  +MOVJ EC00095
SMOVL C00096 BC00096 V=10.0  +MOVJ EC00096
ARCOF
SWVOF
MOVJ C00097 BC00097 VJ=100.00  +MOVJ EC00097 VJ=15.00
SFTOF3D
MOVJ C00098 BC00098 VJ=100.00  +MOVJ EC00098 VJ=100.00
MOVJ C00099 BC00099 VJ=100.00  +MOVJ EC00099 VJ=100.00
MACRO1 MJ#(0) ARGF6
SFTON3D P024
SMOVL C00100 BC00100 V=250.0  +MOVJ EC00100
ARCON
SMOVL C00101 BC00101 V=10.0  +MOVJ EC00101
SMOVL C00102 BC00102 V=12.5  +MOVJ EC00102
SMOVL C00103 BC00103 V=12.5  +MOVJ EC00103
SMOVL C00104 BC00104 V=12.5  +MOVJ EC00104
ARCOF
SFTOF3D
MOVJ C00105 BC00105 VJ=15.00  +MOVJ EC00105 VJ=15.00
MOVJ C00106 BC00106 VJ=100.00  +MOVJ EC00106 VJ=15.00
MACRO1 MJ#(0) ARGF14
MOVJ C00107 BC00107 VJ=20.00  +MOVJ EC00107 VJ=20.00
SFTON3D P023
SMOVL C00108 BC00108 V=133.3  +MOVJ EC00108
ARCON
SMOVL C00109 BC00109 V=10.0  +MOVJ EC00109
SMOVL C00110 BC00110 V=10.0  +MOVJ EC00110
ARCOF
SFTOF3D
MOVJ C00111 BC00111 VJ=15.00  +MOVJ EC00111 VJ=15.00
MOVJ C00112 BC00112 VJ=100.00  +MOVJ EC00112 VJ=15.00
MOVJ C00113 BC00113 VJ=100.00  +MOVJ EC00113 VJ=100.00
SFTON3D P022
SMOVL C00114 BC00114 V=83.3  +MOVJ EC00114
ARCON
SMOVL C00115 BC00115 V=9.2  +MOVJ EC00115
SMOVL C00116 BC00116 V=9.2  +MOVJ EC00116
SMOVL C00117 BC00117 V=11.7  +MOVJ EC00117
SMOVL C00118 BC00118 V=11.7  +MOVJ EC00118
SMOVL C00119 BC00119 V=11.7  +MOVJ EC00119
SMOVL C00120 BC00120 V=11.7  +MOVJ EC00120
SMOVC C00121 BC00121 V=10.0  +MOVJ EC00121
SMOVC C00122 BC00122 V=10.0  +MOVJ EC00122
SMOVC C00123 BC00123 V=10.0  +MOVJ EC00123
SMOVL C00124 BC00124 V=10.0  +MOVJ EC00124
ARCOF
SFTOF3D
MOVJ C00125 BC00125 VJ=15.00  +MOVJ EC00125 VJ=15.00
MOVJ C00126 BC00126 VJ=40.00  +MOVJ EC00126 VJ=15.00
MACRO1 MJ#(0) ARGF6
SFTON3D P021
MOVJ C00127 BC00127 VJ=100.00  +MOVJ EC00127 VJ=40.00
SMOVL C00128 BC00128 V=250.0  +MOVJ EC00128
ARCON
SMOVL C00129 BC00129 V=8.3  +MOVJ EC00129
ARCOF
MOVJ C00130 BC00130 VJ=100.00  +MOVJ EC00130 VJ=100.00
SFTOF3D
MOVJ C00131 BC00131 VJ=100.00  +MOVJ EC00131 VJ=100.00
MOVJ C00132 BC00132 VJ=100.00  +MOVJ EC00132 VJ=100.00
MOVJ C00133 BC00133 VJ=100.00  +MOVJ EC00133 VJ=100.00
SMOVL C00134 BC00134 V=1000.0  +MOVJ EC00134
SFTON3D P071
SMOVL C00135 BC00135 V=400.0  +MOVJ EC00135
SMOVL C00136 BC00136 V=166.7  +MOVJ EC00136
SMOVL C00137 BC00137 V=100.0 PL=0  +MOVJ EC00137
MACRO1 MJ#(0) ARGF9
ARCON
SMOVL C00138 BC00138 V=6.7  +MOVJ EC00138
SWVON WEV#(205)
SMOVL C00139 BC00139 V=6.7  +MOVJ EC00139
ARCOF
SWVOF
SMOVL C00140 BC00140 V=100.0  +MOVJ EC00140
SMOVL C00141 BC00141 V=100.0  +MOVJ EC00141
TIMER T=5.00
SMOVL C00142 BC00142 V=100.0 PL=0  +MOVJ EC00142
SWVON WEV#(205)
ARCON
SMOVL C00143 BC00143 V=5.0  +MOVJ EC00143
ARCOF
SWVOF
SFTOF3D
SMOVL C00144 BC00144 V=400.0  +MOVJ EC00144
SMOVL C00145 BC00145 V=1000.0  +MOVJ EC00145
MOVJ C00146 BC00146 VJ=100.00  +MOVJ EC00146 VJ=100.00
CALL JOB:CLEAN-R1_KM_NEW
MOVJ C00147 BC00147 VJ=100.00  +MOVJ EC00147 VJ=100.00
SFTOF3D
MOVJ C00148 BC00148 VJ=100.00  +MOVJ EC00148 VJ=100.00
MOVJ C00149 BC00149 VJ=100.00  +MOVJ EC00149 VJ=100.00
MOVJ C00150 BC00150 VJ=100.00  +MOVJ EC00150 VJ=100.00
SMOVL C00151 BC00151 V=100.0  +MOVJ EC00151
SREFP 3 C00152 BC00152  +REFP EC00152
CALL JOB:SEARCH-R1-S13D
SET P021 P006
SFTON3D P021
SMOVL C00153 BC00153 V=100.0  +MOVJ EC00153
SREFP 3 C00154 BC00154  +REFP EC00154
CALL JOB:SEARCH-R1-S13D
SET P021 P006
SFTON3D P021
SMOVL C00155 BC00155 V=100.0  +MOVJ EC00155
SFTOF3D
SMOVL C00156 BC00156 V=250.0  +MOVJ EC00156
SMOVL C00157 BC00157 V=100.0  +MOVJ EC00157
SREFP 3 C00158 BC00158  +REFP EC00158
CALL JOB:SEARCH-R1-S13D
SET P022 P006
SFTON3D P022
SMOVL C00159 BC00159 V=100.0  +MOVJ EC00159
SREFP 3 C00160 BC00160  +REFP EC00160
CALL JOB:SEARCH-R1-S13D
SET P022 P006
SFTON3D P022
SMOVL C00161 BC00161 V=100.0  +MOVJ EC00161
SFTOF3D
MOVJ C00162 BC00162 VJ=100.00  +MOVJ EC00162 VJ=100.00
MOVJ C00163 BC00163 VJ=100.00  +MOVJ EC00163 VJ=100.00
MOVJ C00164 BC00164 VJ=100.00  +MOVJ EC00164 VJ=100.00
SMOVL C00165 BC00165 V=100.0  +MOVJ EC00165
SREFP 3 C00166 BC00166  +REFP EC00166
CALL JOB:SEARCH-R1-S13D
SET P023 P006
SFTON3D P023
SMOVL C00167 BC00167 V=100.0  +MOVJ EC00167
SREFP 3 C00168 BC00168  +REFP EC00168
CALL JOB:SEARCH-R1-S13D
SET P023 P006
SFTON3D P023
SMOVL C00169 BC00169 V=100.0  +MOVJ EC00169
SFTOF3D
MOVL C00170 BC00170 V=333.3  +MOVJ EC00170 VJ=100.00
SMOVL C00171 BC00171 V=100.0  +MOVJ EC00171
SREFP 3 C00172 BC00172  +REFP EC00172
CALL JOB:SEARCH-R1-S13D
SET P024 P006
SFTON3D P024
SMOVL C00173 BC00173 V=100.0  +MOVJ EC00173
SREFP 3 C00174 BC00174  +REFP EC00174
CALL JOB:SEARCH-R1-S13D
SET P024 P006
SFTON3D P024
SMOVL C00175 BC00175 V=100.0  +MOVJ EC00175
MOVJ C00176 BC00176 VJ=100.00  +MOVJ EC00176 VJ=100.00
MOVJ C00177 BC00177 VJ=100.00  +MOVJ EC00177 VJ=100.00
MOVJ C00178 BC00178 VJ=100.00  +MOVJ EC00178 VJ=100.00
MOVJ C00179 BC00179 VJ=100.00  +MOVJ EC00179 VJ=100.00
MOVJ C00180 BC00180 VJ=100.00  +MOVJ EC00180 VJ=100.00
SMOVL C00181 BC00181 V=100.0  +MOVJ EC00181
SREFP 3 C00182 BC00182  +REFP EC00182
CALL JOB:SEARCH-R1-S13D
SET P030 P006
SFTON3D P030
SMOVL C00183 BC00183 V=100.0  +MOVJ EC00183
SREFP 3 C00184 BC00184  +REFP EC00184
CALL JOB:SEARCH-R1-S13D
SET P030 P006
SFTON3D P030
SMOVL C00185 BC00185 V=100.0  +MOVJ EC00185
SMOVL C00186 BC00186 V=100.0  +MOVJ EC00186
SREFP 3 C00187 BC00187  +REFP EC00187
CALL JOB:SEARCH-R1-S13D
SET P030 P006
SFTON3D P030
SMOVL C00188 BC00188 V=100.0  +MOVJ EC00188
SFTOF3D
MOVJ C00189 BC00189 VJ=100.00  +MOVJ EC00189 VJ=100.00
MOVJ C00190 BC00190 VJ=100.00  +MOVJ EC00190 VJ=100.00
SMOVL C00191 BC00191 V=100.0  +MOVJ EC00191
SREFP 3 C00192 BC00192  +REFP EC00192
CALL JOB:SEARCH-R1-S13D
SET P031 P006
SFTON3D P031
SMOVL C00193 BC00193 V=100.0  +MOVJ EC00193
SREFP 3 C00194 BC00194  +REFP EC00194
CALL JOB:SEARCH-R1-S13D
SET P031 P006
SFTON3D P031
SMOVL C00195 BC00195 V=100.0  +MOVJ EC00195
SFTOF3D
MOVL C00196 BC00196 V=333.3  +MOVJ EC00196 VJ=100.00
SMOVL C00197 BC00197 V=100.0  +MOVJ EC00197
SREFP 3 C00198 BC00198  +REFP EC00198
CALL JOB:SEARCH-R1-S13D
SET P032 P006
SFTON3D P032
SMOVL C00199 BC00199 V=100.0  +MOVJ EC00199
SREFP 3 C00200 BC00200  +REFP EC00200
CALL JOB:SEARCH-R1-S13D
SET P032 P006
SFTON3D P032
SMOVL C00201 BC00201 V=100.0  +MOVJ EC00201
SFTOF3D
MOVJ C00202 BC00202 VJ=100.00  +MOVJ EC00202 VJ=100.00
MOVJ C00203 BC00203 VJ=100.00  +MOVJ EC00203 VJ=100.00
MOVJ C00204 BC00204 VJ=100.00  +MOVJ EC00204 VJ=100.00
MOVJ C00205 BC00205 VJ=100.00  +MOVJ EC00205 VJ=100.00
MOVJ C00206 BC00206 VJ=100.00  +MOVJ EC00206 VJ=100.00
MOVL C00207 BC00207 V=333.3  +MOVJ EC00207 VJ=100.00
SMOVL C00208 BC00208 V=100.0  +MOVJ EC00208
SREFP 3 C00209 BC00209  +REFP EC00209
CALL JOB:SEARCH-R1-S13D
SET P072 P006
SFTON3D P072
SMOVL C00210 BC00210 V=100.0  +MOVJ EC00210
SMOVL C00211 BC00211 V=100.0  +MOVJ EC00211
SMOVL C00212 BC00212 V=100.0  +MOVJ EC00212
SREFP 3 C00213 BC00213  +REFP EC00213
CALL JOB:SEARCH-R1-S13D
SET P072 P006
SFTON3D P072
SMOVL C00214 BC00214 V=100.0  +MOVJ EC00214
SFTOF3D
SMOVL C00215 BC00215 V=1000.0  +MOVJ EC00215
MOVJ C00216 BC00216 VJ=100.00  +MOVJ EC00216 VJ=100.00
MOVJ C00217 BC00217 VJ=100.00  +MOVJ EC00217 VJ=100.00
SMOVL C00218 BC00218 V=100.0  +MOVJ EC00218
SREFP 3 C00219 BC00219  +REFP EC00219
CALL JOB:SEARCH-R1-S13D
SET P025 P006
SFTON3D P025
SMOVL C00220 BC00220 V=100.0  +MOVJ EC00220
SREFP 3 C00221 BC00221  +REFP EC00221
CALL JOB:SEARCH-R1-S13D
SET P025 P006
SFTON3D P025
SMOVL C00222 BC00222 V=100.0  +MOVJ EC00222
SMOVL C00223 BC00223 V=100.0  +MOVJ EC00223
SREFP 3 C00224 BC00224  +REFP EC00224
CALL JOB:SEARCH-R1-S13D
SET P025 P006
SFTON3D P025
SMOVL C00225 BC00225 V=100.0  +MOVJ EC00225
SFTOF3D
MOVJ C00226 BC00226 VJ=100.00  +MOVJ EC00226 VJ=100.00
MOVJ C00227 BC00227 VJ=100.00  +MOVJ EC00227 VJ=100.00
MOVJ C00228 BC00228 VJ=100.00  +MOVJ EC00228 VJ=100.00
SMOVL C00229 BC00229 V=100.0  +MOVJ EC00229
SREFP 3 C00230 BC00230  +REFP EC00230
CALL JOB:SEARCH-R1-S13D
SET P026 P006
SFTON3D P026
SMOVL C00231 BC00231 V=100.0  +MOVJ EC00231
SREFP 3 C00232 BC00232  +REFP EC00232
CALL JOB:SEARCH-R1-S13D
SET P026 P006
SFTON3D P026
SMOVL C00233 BC00233 V=100.0  +MOVJ EC00233
SMOVL C00234 BC00234 V=100.0  +MOVJ EC00234
SREFP 3 C00235 BC00235  +REFP EC00235
CALL JOB:SEARCH-R1-S13D
SET P026 P006
SFTON3D P026
SMOVL C00236 BC00236 V=100.0  +MOVJ EC00236
SFTOF3D
MOVJ C00237 BC00237 VJ=100.00  +MOVJ EC00237 VJ=100.00
MOVJ C00238 BC00238 VJ=100.00  +MOVJ EC00238 VJ=100.00
MOVJ C00239 BC00239 VJ=100.00  +MOVJ EC00239 VJ=100.00
SMOVL C00240 BC00240 V=100.0  +MOVJ EC00240
SREFP 3 C00241 BC00241  +REFP EC00241
CALL JOB:SEARCH-R1-S13D
SET P027 P006
SFTON3D P027
SMOVL C00242 BC00242 V=100.0  +MOVJ EC00242
SMOVL C00243 BC00243 V=100.0  +MOVJ EC00243
SMOVL C00244 BC00244 V=100.0  +MOVJ EC00244
SREFP 3 C00245 BC00245  +REFP EC00245
CALL JOB:SEARCH-R1-S13D
SET P027 P006
SFTON3D P027
SMOVL C00246 BC00246 V=100.0  +MOVJ EC00246
SREFP 3 C00247 BC00247  +REFP EC00247
CALL JOB:SEARCH-R1-S13D
SET P027 P006
SFTON3D P027
SMOVL C00248 BC00248 V=100.0  +MOVJ EC00248
MOVL C00249 BC00249 V=100.0  +MOVJ EC00249 VJ=100.00
SFTOF3D
MOVJ C00250 BC00250 VJ=100.00  +MOVJ EC00250 VJ=100.00
SMOVL C00251 BC00251 V=100.0  +MOVJ EC00251
SREFP 3 C00252 BC00252  +REFP EC00252
CALL JOB:SEARCH-R1-S13D
SET P028 P006
SFTON3D P028
SMOVL C00253 BC00253 V=100.0  +MOVJ EC00253
SMOVL C00254 BC00254 V=100.0  +MOVJ EC00254
SREFP 3 C00255 BC00255  +REFP EC00255
CALL JOB:SEARCH-R1-S13D
SET P028 P006
SFTON3D P028
SMOVL C00256 BC00256 V=100.0  +MOVJ EC00256
SMOVL C00257 BC00257 V=100.0  +MOVJ EC00257
SREFP 3 C00258 BC00258  +REFP EC00258
CALL JOB:SEARCH-R1-S13D
SET P028 P006
SFTON3D P028
SMOVL C00259 BC00259 V=100.0  +MOVJ EC00259
MOVJ C00260 BC00260 VJ=100.00  +MOVJ EC00260 VJ=100.00
MOVJ C00261 BC00261 VJ=100.00  +MOVJ EC00261 VJ=100.00
MOVJ C00262 BC00262 VJ=100.00  +MOVJ EC00262 VJ=100.00
MACRO1 MJ#(0) ARGF14
SMOVL C00263 BC00263 V=133.3  +MOVJ EC00263
ARCON
SMOVL C00264 BC00264 V=10.0  +MOVJ EC00264
ARCOF
MOVJ C00265 BC00265 VJ=100.00  +MOVJ EC00265 VJ=100.00
SFTOF3D
MOVJ C00266 BC00266 VJ=100.00  +MOVJ EC00266 VJ=100.00
MOVJ C00267 BC00267 VJ=100.00  +MOVJ EC00267 VJ=100.00
SFTON3D P027
SMOVL C00268 BC00268 V=133.3  +MOVJ EC00268
ARCON
SMOVL C00269 BC00269 V=10.0  +MOVJ EC00269
SMOVL C00270 BC00270 V=10.0  +MOVJ EC00270
SMOVL C00271 BC00271 V=10.8  +MOVJ EC00271
SMOVL C00272 BC00272 V=11.7  +MOVJ EC00272
SMOVC C00273 BC00273 V=11.7  +MOVJ EC00273
SMOVC C00274 BC00274 V=10.0  +MOVJ EC00274
SMOVC C00275 BC00275 V=10.0  +MOVJ EC00275
SMOVL C00276 BC00276 V=10.0  +MOVJ EC00276
ARCOF
MOVJ C00277 BC00277 VJ=100.00  +MOVJ EC00277 VJ=100.00
MOVJ C00278 BC00278 VJ=100.00  +MOVJ EC00278 VJ=100.00
SFTOF3D
MOVJ C00279 BC00279 VJ=100.00  +MOVJ EC00279 VJ=100.00
SFTON3D P026
SMOVL C00280 BC00280 V=133.3  +MOVJ EC00280
ARCON
SMOVL C00281 BC00281 V=10.0  +MOVJ EC00281
SMOVL C00282 BC00282 V=10.0  +MOVJ EC00282
SMOVL C00283 BC00283 V=10.0  +MOVJ EC00283
SMOVL C00284 BC00284 V=10.0  +MOVJ EC00284
ARCOF
MOVJ C00285 BC00285 VJ=100.00  +MOVJ EC00285 VJ=100.00
MOVJ C00286 BC00286 VJ=100.00  +MOVJ EC00286 VJ=100.00
SFTON3D P025
MOVJ C00287 BC00287 VJ=100.00  +MOVJ EC00287 VJ=100.00
MACRO1 MJ#(0) ARGF6
SMOVL C00288 BC00288 V=133.3  +MOVJ EC00288
ARCON
SMOVL C00289 BC00289 V=10.0  +MOVJ EC00289
SMOVL C00290 BC00290 V=10.0  +MOVJ EC00290
SMOVL C00291 BC00291 V=10.0  +MOVJ EC00291
SMOVL C00292 BC00292 V=10.0  +MOVJ EC00292
SMOVL C00293 BC00293 V=10.0  +MOVJ EC00293
ARCOF
SFTOF3D
MOVJ C00294 BC00294 VJ=100.00  +MOVJ EC00294 VJ=100.00
MOVJ C00295 BC00295 VJ=100.00  +MOVJ EC00295 VJ=100.00
MOVJ C00296 BC00296 VJ=100.00  +MOVJ EC00296 VJ=100.00
MOVJ C00297 BC00297 VJ=100.00  +MOVJ EC00297 VJ=100.00
SMOVL C00298 BC00298 V=166.7  +MOVJ EC00298
SFTON3D P072
SMOVL C00299 BC00299 V=100.0 PL=0  +MOVJ EC00299
MACRO1 MJ#(0) ARGF9
ARCON
SMOVL C00300 BC00300 V=6.7  +MOVJ EC00300
SWVON WEV#(205)
SMOVL C00301 BC00301 V=6.7  +MOVJ EC00301
ARCOF
SWVOF
SMOVL C00302 BC00302 V=166.7  +MOVJ EC00302
SMOVL C00303 BC00303 V=166.7  +MOVJ EC00303
TIMER T=5.00
SMOVL C00304 BC00304 V=100.0 PL=0  +MOVJ EC00304
SWVON WEV#(205)
SMOVL C00305 BC00305 V=5.0  +MOVJ EC00305
ARCOF
SWVOF
SMOVL C00306 BC00306 V=166.7  +MOVJ EC00306
SFTOF3D
MOVL C00307 BC00307 V=1000.0  +MOVJ EC00307 VJ=100.00
MOVJ C00308 BC00308 VJ=100.00  +MOVJ EC00308 VJ=100.00
MOVJ C00309 BC00309 VJ=100.00  +MOVJ EC00309 VJ=100.00
MOVJ C00310 BC00310 VJ=100.00  +MOVJ EC00310 VJ=100.00
MOVJ C00311 BC00311 VJ=100.00  +MOVJ EC00311 VJ=100.00
MACRO1 MJ#(0) ARGF14
MOVJ C00312 BC00312 VJ=100.00  +MOVJ EC00312 VJ=100.00
SFTON3D P023
SMOVL C00313 BC00313 V=133.3  +MOVJ EC00313
ARCON
SWVON WEV#(14)
SFTON3D P024
SMOVL C00314 BC00314 V=7.5  +MOVJ EC00314
ARCOF
SWVOF
MOVJ C00315 BC00315 VJ=100.00  +MOVJ EC00315 VJ=100.00
MOVJ C00316 BC00316 VJ=100.00  +MOVJ EC00316 VJ=100.00
MOVJ C00317 BC00317 VJ=100.00  +MOVJ EC00317 VJ=100.00
MOVJ C00318 BC00318 VJ=100.00  +MOVJ EC00318 VJ=100.00
SFTON3D P021
SMOVL C00319 BC00319 V=133.3  +MOVJ EC00319
SREFP 1 C00320 BC00320  +REFP EC00320
SREFP 2 C00321 BC00321  +REFP EC00321
ARCON
SWVON WEV#(14)
SFTON3D P022
SMOVL C00322 BC00322 V=7.5  +MOVJ EC00322
ARCOF
SWVOF
MOVJ C00323 BC00323 VJ=100.00  +MOVJ EC00323 VJ=100.00
MOVJ C00324 BC00324 VJ=100.00  +MOVJ EC00324 VJ=100.00
MOVJ C00325 BC00325 VJ=100.00  +MOVJ EC00325 VJ=100.00
MOVJ C00326 BC00326 VJ=100.00  +MOVJ EC00326 VJ=100.00
MOVJ C00327 BC00327 VJ=100.00  +MOVJ EC00327 VJ=100.00
MOVJ C00328 BC00328 VJ=100.00  +MOVJ EC00328 VJ=100.00
MOVJ C00329 BC00329 VJ=100.00  +MOVJ EC00329 VJ=100.00
MACRO1 MJ#(0) ARGF9
SFTON3D P030
SMOVL C00330 BC00330 V=133.3 PL=0  +MOVJ EC00330
SREFP 1 C00331 BC00331  +REFP EC00331
SREFP 2 C00332 BC00332  +REFP EC00332
SWVON WEV#(68)
ARCON
SMOVL C00333 BC00333 V=10.0  +MOVJ EC00333
SMOVL C00334 BC00334 V=10.0  +MOVJ EC00334
SMOVL C00335 BC00335 V=10.0  +MOVJ EC00335
COMM SMOVL C00336 BC00336 V=10.0  +MOVJ EC00336
ARCOF
SWVOF
MOVJ C00337 BC00337 VJ=100.00  +MOVJ EC00337 VJ=100.00
MOVJ C00338 BC00338 VJ=100.00  +MOVJ EC00338 VJ=100.00
SMOVL C00339 BC00339 V=133.3 PL=0  +MOVJ EC00339
ARCON
SWVON WEV#(61)
SMOVL C00340 BC00340 V=8.3  +MOVJ EC00340
ARCOF
SWVOF
MOVJ C00341 BC00341 VJ=100.00  +MOVJ EC00341 VJ=100.00
MOVJ C00342 BC00342 VJ=100.00  +MOVJ EC00342 VJ=100.00
SFTON3D P032
MOVJ C00343 BC00343 VJ=100.00  +MOVJ EC00343 VJ=100.00
MACRO1 MJ#(0) ARGF9
SMOVL C00344 BC00344 V=133.3  +MOVJ EC00344
ARCON
SMOVL C00345 BC00345 V=8.3  +MOVJ EC00345
SFTON3D P031
SWVON WEV#(61)
SMOVL C00346 BC00346 V=10.0  +MOVJ EC00346
SMOVL C00347 BC00347 V=10.0  +MOVJ EC00347
SMOVL C00348 BC00348 V=10.0  +MOVJ EC00348
ARCOF
SWVOF
MOVJ C00349 BC00349 VJ=100.00  +MOVJ EC00349 VJ=100.00
SFTOF3D
MOVJ C00350 BC00350 VJ=100.00  +MOVJ EC00350 VJ=100.00
MOVJ C00351 BC00351 VJ=100.00  +MOVJ EC00351 VJ=100.00
MOVJ C00352 BC00352 VJ=100.00  +MOVJ EC00352 VJ=100.00
MOVJ C00353 BC00353 VJ=100.00  +MOVJ EC00353 VJ=100.00
MOVJ C00354 BC00354 VJ=100.00  +MOVJ EC00354 VJ=100.00
MOVJ C00355 BC00355 VJ=100.00  +MOVJ EC00355 VJ=100.00
MOVJ C00356 BC00356 VJ=100.00  +MOVJ EC00356 VJ=100.00
MACRO1 MJ#(0) ARGF9
SFTON3D P023
SMOVL C00357 BC00357 V=133.3  +MOVJ EC00357
SREFP 2 C00358 BC00358  +REFP EC00358
SREFP 1 C00359 BC00359  +REFP EC00359
ARCON
SWVON WEV#(14)
SMOVL C00360 BC00360 V=8.3  +MOVJ EC00360
ARCOF
SWVOF
MOVJ C00361 BC00361 VJ=100.00  +MOVJ EC00361 VJ=100.00
MOVJ C00362 BC00362 VJ=100.00  +MOVJ EC00362 VJ=100.00
SFTON3D P021
SMOVL C00363 BC00363 V=133.3  +MOVJ EC00363
ARCON
SWVON WEV#(14)
SMOVL C00364 BC00364 V=8.3  +MOVJ EC00364
ARCOF
SWVOF
SFTOF3D
MOVJ C00365 BC00365 VJ=100.00  +MOVJ EC00365 VJ=100.00
MOVJ C00366 BC00366 VJ=100.00  +MOVJ EC00366 VJ=100.00
MOVJ C00367 BC00367 VJ=100.00  +MOVJ EC00367 VJ=100.00
MOVJ C00368 BC00368 VJ=100.00  +MOVJ EC00368 VJ=100.00
MOVJ C00369 BC00369 VJ=100.00  +MOVJ EC00369 VJ=100.00
MOVJ C00370 BC00370 VJ=100.00  +MOVJ EC00370 VJ=100.00
'KONIEC
END
